{attribute 'GeneratedUsingTerminal: EPP3174-0002-0016'}
{attribute addProperty BoxType "EPP3174-0002-0016"}
{attribute addProperty Id "StatusAT %I*Status_B07533568ValueAT %I*INT2"}
{attribute addProperty CRC "2833212643"}
{attribute addProperty Size "10"}
TYPE AI_Standard_Channel_A8DF64E3 :
STRUCT
	{attribute addProperty Name "Status"}
	Status AT %I* : Status_B0753356;
	{attribute addProperty Name "Value"}
	Value AT %I* : INT;
END_STRUCT
END_TYPE

(* stored: Version 1.2.0.0, ProductVersion 3.1.4024.9
   DUT AI_Standard_Channel_A8DF64E3: Id {0e330eff-4f3f-488d-9809-060d11d61c08} *)
